{attribute 'linkalways'} 
{attribute 'no_explicit_call' := 'This FB is a CLASS and must be accessed using methods or properties'}
{attribute 'enable_dynamic_creation'}
FUNCTION_BLOCK FINAL GT_USINT EXTENDS Node
VAR
	in1 : _USINT(0);
	in2 : _USINT(0);
	out : _BOOL(FALSE);
END_VAR

METHOD PUBLIC Clone : I_Node
VAR
	pNode : POINTER TO GT_USINT;
END_VAR
pNode := __NEW(GT_USINT);
Clone := pNode^;
END_METHOD

METHOD FB_init : BOOL
VAR_INPUT
	bInitRetains : BOOL; // if TRUE, the retain variables are initialized (warm start / cold start)
	bInCopyCode : BOOL;  // if TRUE, the instance afterwards gets moved into the copy code (online change)
END_VAR
AddInput('in1',THIS^.in1);
AddInput('in2',THIS^.in2);
AddOutput('out', THIS^.out);
END_METHOD

METHOD PROTECTED OnExecute
VAR
END_VAR
out.Value := in1.Value > in2.Value;
END_METHOD

END_FUNCTION_BLOCK

(* stored: Version 1.1.0.1, ProductVersion 3.1.4024.15
   POU GT_USINT: Id {10fa73d3-ce3b-4f75-b9b1-ffb67067efdb}, SpecialFunc None
   Folder Constructor: Id {716df055-0483-4529-ba5c-abf9cb471049}
   Method Clone: Id {e5c589a2-aea5-441c-85d8-e34bee0173bf}
   Method FB_init: Id {ed34d8f1-5262-44c3-a927-b6fbbb411dbc}
   Method OnExecute: Id {5079baa7-d76b-48eb-9123-6d754633dff4} *)
